METHOD parktelescope: USINT
VAR_INPUT
END_VAR
VAR
	ParkEvent:	FB_Eventlog;
	command_timeout:	TON;
END_VAR
VAR_STAT
	Stage:		USINT := 0;
	LastStage:	USINT := 101;
END_VAR
parktelescope := Stage;
command_timeout(IN := Stage < 100, PT := T#600S);
IF command_timeout.Q THEN
	error := TRUE;
	errorid := 16#20;
	Stage := 0;
END_IF
IF reset OR error THEN
	Stage := 0;
END_IF
IF isparked THEN
	Stage := 100;
END_IF
CASE Stage OF
	0: 
		gohome := 	FALSE;
		track := 	FALSE;
		goto := 	FALSE;
		slew := 	FALSE;
		IF Error THEN // emergency park
			HydraulicsControl.close_brake();
			ElevationControl.enable := FALSE;
			AzimuthElevationControl.Enable := FALSE;
			CoverControl.close := TRUE;	
			Stage := 80;
		END_IF
		Stage := 20;
	20:
		ElevationControl.position := elevation_park;
		ElevationControl.velocity := 10.0;
		ElevationControl.MoveAxis := TRUE;
		AzimuthElevationControl.position := azimuth_park;
		AzimuthElevationControl.velocity := 10;
		AzimuthElevationControl.MoveAxis := TRUE;
		IF ElevationControl.ElevationAxis.Busy AND
			AzimuthElevationControl.AzimuthAxis.Busy THEN
				Stage := 40;
		END_IF
	40:
		IF ElevationControl.ElevationAxis.MoveDone THEN
			ElevationControl.MoveAxis := FALSE;
		END_IF
		IF AzimuthElevationControl.AzimuthAxis.MoveDone THEN
			AzimuthElevationControl.MoveAxis := FALSE;
		END_IF
		IF NOT sliding THEN // all axis standstill
			Stage := 60;
		END_IF
	60:
		IF stopped THEN 
			ElevationControl.enable := FALSE;
			AzimuthElevationControl.Enable := FALSE;
			Stage := 80;
		END_IF
		
		ElevationControl.MoveAxis := FALSE;
		AzimuthElevationControl.MoveAxis := FALSE;
	80:
		IF HydraulicsControl.brake_closed THEN
			CoverControl.close := TRUE;			
		END_IF
		IF CoverControl.isclosed THEN
			Stage := 100;
		END_IF
	100:
			isparked := TRUE;
			park := FALSE;
			parktelescope := 100;
			Stage := 0;	
END_CASE
ParkEvent(Trigger := Stage > LastStage, FormatString := 'Parking progress: %s', OnMessage := USINT_TO_STRING(Stage));
LastStage := Stage;
END_METHOD

METHOD poweron : BOOL
VAR_INPUT
END_VAR
VAR
END_VAR
IF NOT Main.brake_clearing THEN
	powerfailure := TRUE;
	TCSpowerEvent.OnMessage := 'failure: brake clearing not set';
	power := FALSE;
ELSIF NOT Transformer.power_OK THEN
	powerfailure := TRUE;
	TCSpowerEvent.OnMessage := 'failure: main power failure';
	power := FALSE;
ELSIF NOT Transformer.phase_available THEN
	powerfailure := TRUE;
	TCSpowerEvent.OnMessage := 'failure: hydraulics power failure';
	power := FALSE;
ELSIF error THEN
	powerfailure := TRUE;
	TCSpowerEvent.OnMessage := 'Generic error during power on occured.';
	power := FALSE;
ELSE
	powerfailure := FALSE;		
END_IF
// COVER MUST BE OPENED FOR A SUCCESSFUL WAKE & SHAKE COMMAND!
Covercontrol.open := TRUE;

// enable elevation, enable azimuth
IF MAIN.ready AND CoverControl.isopen THEN
	ElevationControl.enable := TRUE;
	AzimuthElevationControl.enable := TRUE;
END_IF

IF ElevationControl.Ready AND NOT ElevationControl.Calibrated THEN
	ElevationControl.HomeAxis := TRUE;
END_IF

IF AzimuthElevationControl.ready AND NOT AzimuthElevationControl.calibrated THEN
	AzimuthElevationControl.HomeAxis := TRUE;
END_IF

// start calibration of focus after elevation has been calibrated
// this avoids imbalance by the M2 mirror on the elvation during its calibration

IF CoverControl.isopen AND 
	ElevationControl.Calibrated AND ElevationControl.Ready AND
	AzimuthElevationControl.calibrated AND AzimuthElevationControl.ready THEN
	power := FALSE;
	poweron := TRUE;
	isparked := FALSE;
	// slew the telescope to the home position
	gohome := TRUE;
ELSE
	poweron := FALSE;
END_IF
END_METHOD

METHOD slewtelescope : USINT
VAR_INPUT
END_VAR
VAR
	SlewEvent:	FB_Eventlog;
	command_timeout: TON;
END_VAR
VAR_STAT
	Stage:		USINT := 0;
	LastStage:	USINT := 101;
END_VAR
slewtelescope := Stage;
command_timeout(IN := Stage < 100, PT := T#600S);
IF command_timeout.Q THEN
	error := TRUE;
	errorid := 16#40;
	slew := FALSE;
	Stage := 0;
END_IF
IF reset OR error THEN
	Stage := 0;
END_IF
CASE Stage OF
	0:	
		IF ready AND stopped AND NOT busy AND NOT tracking THEN
			Stage := 25;
		END_IF
	25:
		ElevationControl.position := elevation;
		ElevationControl.velocity := 5.0;
		ElevationControl.MoveAxis := TRUE;
		AzimuthElevationControl.position := azimuth;
		AzimuthElevationControl.velocity := 10.0;
		AzimuthElevationControl.MoveAxis := TRUE;
		IF ElevationControl.ElevationAxis.Busy AND
			AzimuthElevationControl.AzimuthAxis.Busy THEN
				Stage := 50;
		END_IF
	50:
		IF ElevationControl.ElevationAxis.MoveDone THEN
			ElevationControl.MoveAxis := FALSE;
		END_IF
		
		IF AzimuthElevationControl.AzimuthAxis.MoveDone THEN
			AzimuthElevationControl.MoveAxis := FALSE;
		END_IF

		IF NOT sliding AND stopped THEN // all axis standstill
			Stage := 100;
		END_IF
	100:
		ElevationControl.MoveAxis := FALSE;
		AzimuthElevationControl.MoveAxis := FALSE;
		rightascension := rightascension_calc;
		declination := declination_calc;
		slew := FALSE;
		Stage := 0;
END_CASE
SlewEvent(Trigger := Stage > LastStage, FormatString := 'Slew progress: %s', OnMessage := USINT_TO_STRING(Stage));
LastStage := Stage;
END_METHOD

METHOD stoptelescope : BOOL
VAR_INPUT
END_VAR
ElevationControl.StopAxis := TRUE;
AzimuthElevationControl.StopAxis := TRUE;
IF stopped THEN
	ElevationControl.StopAxis := FALSE;
	AzimuthElevationControl.StopAxis := FALSE;
	stop := FALSE;
END_IF
END_METHOD

METHOD tracktelescope : BOOL
VAR_INPUT
END_VAR
// Elevation
ElevationVelocity := F_Elevationvelocity(azimuth_calc, latitude);
AzimuthVelocity := F_Azimuthvelocity(elevation_calc, azimuth_calc, latitude);
IF elevation_current < 5.0 OR elevation_current > 89.5 THEN 
	track := FALSE;
END_IF
IF azimuth_current > 440.0 THEN
	track := FALSE;
END_IF

ElevationControl.position := elevation_calc;
IF NOT ElevationControl.Tracking THEN
	ElevationControl.velocity := 10.0;
	ElevationControl.MoveAxis := TRUE;
	IF NOT ElevationControl.ElevationAxis.Busy AND ElevationControl.ElevationAxis.MoveDone THEN
		ElevationControl.MoveAxis := FALSE;
		IF ElevationControl.ElevationAxis.isTracking THEN
			ElevationControl.velocity := ElevationVelocity;
		ELSE
			ElevationControl.velocity := 3.0*ElevationVelocity;
		END_IF
		ElevationControl.velocity := ElevationVelocity;
		ElevationControl.Tracking := TRUE;
	END_IF
ELSE
	ElevationControl.velocity := ElevationVelocity;
END_IF

// Azimuth
AzimuthElevationControl.position := azimuth_calc;
IF NOT AzimuthElevationControl.Tracking THEN
	AzimuthElevationControl.velocity := 10.0;
	AzimuthElevationControl.MoveAxis := TRUE;
	IF NOT AzimuthElevationControl.AzimuthAxis.Busy AND AzimuthElevationControl.AzimuthAxis.MoveDone THEN
		AzimuthElevationControl.MoveAxis := FALSE;
		IF AzimuthElevationControl.AzimuthAxis.isTracking THEN
			AzimuthElevationControl.velocity := AzimuthVelocity;
		ELSE
			AzimuthElevationControl.velocity := 3.0*AzimuthVelocity;
		END_IF
		AzimuthElevationControl.velocity := AzimuthVelocity;
		AzimuthElevationControl.Tracking := TRUE;
	END_IF
ELSE
	AzimuthElevationControl.velocity := AzimuthVelocity;
END_IF
END_METHOD

END_PROGRAM

// ---- POUs/Function Blocks/FB_EQ2HOR2.TcPOU
FUNCTION_BLOCK FB_EQ2HOR2
VAR_INPUT
	// right ascension in degrees
	alpha: LREAL;
	// declination in degrees
	delta: LREAL;
	// longitude in degrees
	lon: LREAL;
	// latitude in degrees
	lat: LREAL;
	// Julian Days
	JD: LREAL;
END_VAR
VAR_OUTPUT
	// altitude in degrees
	alt: LREAL;
	// azimuth in degrees
	az: LREAL;
	// hour angle in degreesss
	ha: LREAL;
END_VAR
VAR
	lst: LREAL;
	// helper variables
	sinalt,
	// in radians
	phi_r, tau_r, alpha_r, delta_r: LREAL;
	// current epoch
	J_now: 		LREAL;
	// enable precession
	precess: 	BOOL := TRUE;
	// enable nutation
	nutate:		BOOL := TRUE;
	// enable abberation
	abberation:	BOOL := TRUE;
	// enable refraction correction
	refract:	BOOL := TRUE;
	// precession function block
	fbprecess: 	FB_PRECESS3;
	// nutation function block
	co_nutate: CO_NUTATE;
	// abberration function block
	fbaberration: CO_ABERRATION;
	//precessed coordinates
	alpha1, delta1, 
	d_alpha2, d_delta2, 
	d_alpha3, d_delta3:	LREAL;
END_VAR
VAR CONSTANT
	d2r:	LREAL := PI/180.0;
	r2d:	LREAL := 180.0/PI;
END_VAR

(* 
source: http://star-www.st-and.ac.uk/~fv/webnotes/chapter7.htm
https://squarewidget.com/astronomical-calculations-sidereal-time/

*)
lst := ct2lst(lon, jd) * 15.0; // lst in degrees

J_now := (JD - 2451545.0)/365.25 + 2000.0; // compute current equinox
IF precess THEN
	fbprecess( ra := alpha, dec := delta, 
	//EQUINOX1 := 2000.0, EQUINOX2 := J_now, 
	ra_precessed =>alpha1, dec_precessed => delta1);
ELSE
	alpha1 := alpha;
	delta1 := delta;	
END_IF

IF nutate THEN
	co_nutate(	jd := jd, 
				ra := alpha, 
				dec := delta, 
				d_ra => d_alpha2, 
				d_dec => d_delta2);
	alpha1 := alpha1 + d_alpha2;
	delta1 := delta1 + d_delta2;
ELSE
	d_alpha2 := 0.0;
	d_delta2 := 0.0;
END_IF

IF abberation THEN
	fbaberration(	jd := jd, 
					ra := alpha, 
					dec := delta, 
					d_ra => d_alpha3, 
					d_dec => d_delta3);
	alpha1 := alpha1 + d_alpha3;
	delta1 := delta1 + d_delta3;
ELSE
	d_alpha3 := 0.0;
	d_delta3 := 0.0;
END_IF

ha := MODABS(lst - alpha1, 360.0);

alpha_r := alpha1 * d2r;
delta_r := delta1 * d2r;
tau_r := lst*d2r - alpha_r;
phi_r := lat*d2r;

sinalt := SIN(phi_r)*SIN(delta_r) + COS(phi_r)*COS(delta_r)*COS(tau_r);
alt := ASIN(sinalt) * r2d;
IF refract THEN
	alt := alt + Refraction(alt, pressure := 770.0, temperature := 10.0);
END_IF
az := ATAN2(SIN(tau_r), SIN(phi_r)*COS(tau_r) - COS(phi_r)*TAN(delta_r)) * r2d + 180.0;

END_FUNCTION_BLOCK

// ---- POUs/Function Blocks/CO_ABERRATION.TcPOU
FUNCTION_BLOCK CO_ABERRATION
VAR_INPUT
	jd, 				// Julian Date
	ra, dec: LREAL; 	//ra and dec in degrees
	eps : LREAL := 0.0;
END_VAR
VAR_OUTPUT
	d_ra, d_dec: LREAL;
END_VAR
VAR
	sunpos: FB_SUNPOS;
	nutate: FB_NUTATE;
	sunra, sundec, sunlon,
	d_psi, d_epsilon, eps0,
	t, e, peri, cd, sd, ce, te, cp, sp, cs, ss, ca, sa, term1, term2, term3, term4: LREAL;
END_VAR
VAR CONSTANT
	d2r : LREAL := PI/180.0;
	k: LREAL := 20.49552; //constant of aberration, in arcseconds
	
END_VAR

(*
;+
;  NAME:
;     CO_ABERRATION
; PURPOSE:
;     Calculate changes to Ra and Dec due to the effect of annual aberration 
; EXPLANATION:
;      as described in Meeus, Chap 23.
; CALLING SEQUENCE:
;      co_aberration, jd, ra, dec, d_ra, d_dec, [EPS = ]
; INPUTS
;       jd      : Julian Date [scalar or vector]
;       ra, dec : Arrays (or scalars) of the ra  and dec's in degrees
;   Note: if jd is a vector, then ra and dec must either be scalars, or 
;                vectors of the same length.
;
; OUTPUTS
;       d_ra, d_dec: the corrections to ra and dec due to aberration in 
;                    arcseconds.  (These values can be added to the true RA 
;                    and dec to get the apparent position).   Note that d_ra
;                     is *not* multiplied by cos(dec), so that 
;                     apparent_ra = ra + d_ra/3600. 
; OPTIONAL INPUT KEYWORD:
;       eps : set this to the true obliquity of the ecliptic (in radians), or
;         it will be set for you if you don't know it (in that case, set it to
;                 an empty variable).
; EXAMPLE:
;   Compute the change in RA and Dec of Theta Persei (RA = 2h46m,11.331s, Dec =
;   49d20',54.54") due to aberration on 2028 Nov 13.19 TD
;
;      IDL> jdcnv,2028,11,13,.19*24,jd      ;Get Julian date
;      IDL> co_aberration,jd,ten(2,46,11.331)*15,ten(49,20,54.54),d_ra,d_dec
;
;      ==> d_ra = 30.045" (=2.003s)    d_dec = 6.697"
; NOTES:
;  These formula are from Meeus, Chapters 23.  Accuracy is much better than 1 
;   arcsecond.
;
;   The maximum deviation due to annual aberration is 20.49" and occurs when the
;   Earth velocity is perpendicular to the direction of the star.
;
; REVISION HISTORY:
;   Written, June 2002,      Chris O'Dell, U. of Wisconsin
;   Fix error with vector input   W. Landsman   June 2009
;   June 2009 update fixed case where JD was scalar but RA,Dec were vectors, but 
;     broke the case when both JD and RA,Dec were vectors Aug 2012 W. Landsman
;   Further fix when JD is 1 element vector  W. Landsman
;-
*)

T := (jd -2451545.0)/36525.0; // julian centuries from J2000 of jd.

IF EPS = 0.0 THEN
	// must calculate obliquity of ecliptic
	nutate(jd := jd, nut_long => d_psi, nut_obliq => d_epsilon); //d_psi and d_epsilon in degrees
	eps0 := ten(23,26,21.448)*3600.0 - 46.8150*T - 0.00059*EXPT(T, 2) +  0.001813*EXPT(T, 3);
	// TRUE obliquity OF the ecliptic in radians
	eps := (eps0 + d_epsilon)/3600.0*d2r; 	
END_IF

sunpos( JD := jd, RA => sunra, Dec => sundec, longmed => sunlon);

// Earth's orbital eccentricity
e := 0.016708634 - 0.000042037*T - 0.0000001267*EXPT(T, 2);
// longitude of perihelion, in degrees 
peri := 102.93735 + 1.71946*T + 0.00046*EXPT(T, 2);

//Useful Trig Functions
cd := COS(dec*d2r);		sd := SIN(dec*d2r);
ce := COS(eps); 		te := TAN(eps);
cp := COS(peri*d2r);	sp := SIN(peri*d2r);
cs := COS(sunlon*d2r);	ss := SIN(sunlon*d2r);
ca := COS(ra*d2r);		sa := SIN(ra*d2r);

term1 := (ca*cs*ce + sa*ss)/cd;
term2 := (ca*cp*ce + sa*sp)/cd;
term3 := (cs*ce*(te*cd - sa*sd) + ca*sd*ss);
term4 := (cp*ce*(te*cd - sa*sd) + ca*sd*sp);

d_ra := (-k * term1 + e*k * term2)/3600.0;
d_dec := (-k * term3 + e*k * term4)/3600.0;

END_FUNCTION_BLOCK

// ---- POUs/Functions/Refraction.TcPOU
FUNCTION Refraction : LREAL
VAR_INPUT
	// elevation in degrees
	elevation: LREAL;
	// pressure in mBar
	pressure: LREAL := 770.0;
	// temperature in Celsius
	temperature : LREAL := 10.0;
END_VAR
VAR
END_VAR
VAR CONSTANT
	d2r:	LREAL := PI/180.0;
END_VAR

// sanity checks
elevation := LIMIT(0.0, elevation, 90.0);
pressure := LIMIT(600.0, pressure, 1200.0);
temperature := LIMIT(-30.0, temperature, 40.0);
// refraction in arcmin
Refraction := 1.02 / TAN((elevation + 10.3/(elevation + 5.11)) * d2r);
Refraction := Refraction * pressure * 283.0 / (1010.0 * (273.0 + temperature));
//refraction in degrees
Refraction := Refraction / 60.0;

END_FUNCTION

// ---- POUs/Function Blocks/FB_HOR2EQ.TcPOU
FUNCTION_BLOCK FB_HOR2EQ
VAR_INPUT
	//altitude (in degrees) [scalar OR vector]
	alt: LREAL;  
	//azimuth angle (in degrees, measured EAST from NORTH, but see keyword WS below.) [scalar or vector]
	az: LREAL;
	// Julian Date [scalar or vector], double precision
	JD: 		LREAL;
	lat:		LREAL;
	lon:		LREAL;
	WS:			BOOL;
	precess:	BOOL := FALSE;
	NUTATE:		BOOL := FALSE;
	aberration:	BOOL := FALSE;
	refract:	BOOL := FALSE;
	altitude:	LREAL := 0.0;
END_VAR
VAR_OUTPUT
	// Right Ascension of object  (J2000) in degrees (FK5)
	ra: 	LREAL;
	// Declination of object (J2000) in degrees (FK5)
	dec:	LREAL;
	// hour angle (in degrees) (optional)
	ha:		LREAL;
END_VAR
VAR
	
	alt_,
	az_,
	lmst,
	J_now: LREAL;
	co_nutate: 		FB_CO_NUTATE;
	co_aberration: 	CO_ABERRATION;
	co_refract:		CO_REFRACT;
	fbprecess:		FB_PRECESS;
	altaz2hadec:	FB_ALTAZ2HADEC;
	last: LREAL;
	dra1: LREAL;
	ddec1: LREAL;
	eps: LREAL;
	d_psi: LREAL;
	dra2: LREAL;
	ddec2: LREAL;
END_VAR
VAR CONSTANT
	//d2r:	LREAL := PI/180.0;
	//r2d:	LREAL := 180.0/PI;
	//h2r:	LREAL := PI/12.0;
	h2d:	LREAL := 15.0;
END_VAR

alt_ := alt;   //do this so we don't change ra, dec arrays.
az_ := az;


//*******************************************************************************************
// Make Correction for ATMOSPHERIC REFRACTION
// (use this for visible and radio wavelengths; author is unsure about other wavelengths)
IF refract THEN 
	co_refract(	old_alt := alt, 
				altitude := altitude, 
				to_observed := TRUE, 
				new_alt => alt);
END_IF

IF WS THEN 
	az_ := az_ - 180.0;
END_IF

co_nutate(	jd := jd, 
			ra := 45.0, 
			dec := 45.0, 
			d_ra => dra1, 
			d_dec => ddec1, 
			eps => eps, 
			d_psi => d_psi);
//******************************************************************************
//Calculate LOCAL APPARENT SIDEREAL TIME
// first get local mean sidereal time (lmst)
// get LST (in hours) - note:this is indep of tzone since giving jd
lmst := ct2lst( lon, jd);
// convert LMST TO degrees (btw, THIS is the RA OF the zenith)
lmst := lmst*h2d;
// calculate local APPARENT sidereal time (last)
// ADD correction in degrees
last := lmst + d_psi *COS(eps)/3600.0 ; 

//****************************************************************************
// Now do the spherical trig to get APPARENT Hour Angle [degrees], and
// declination [degrees].
altaz2hadec( alt := alt_, az := az_, lat := lat, ha => ha, dec => dec);

// Find Right Ascension (in degrees, from 0 to 360.)
 ra := MODABS(last - ha + 360.0, 360.0);



//*****************************************************************************
// calculate NUTATION and ABERRATION Corrections to Ra-Dec
IF NUTATE THEN
	co_nutate(	jd := jd, 
			ra := ra, 
			dec := dec, 
			d_ra => dra1, 
			d_dec => ddec1, 
			eps => eps, 
			d_psi => d_psi);
ELSE
	dra1 := 0.0;
	ddec1 := 0.0;	
END_IF
IF aberration THEN
	co_aberration(	jd := jd, 
				ra := ra, 
				dec := dec, 
				d_ra => dra2, 
				d_dec => ddec2, 
				eps := eps);
ELSE
	dra2 := 0.0;
	ddec2 := 0.0;	
END_IF
//******************************************************************************
// Make Nutation and Aberration Corrections (if wanted)

ra := ra - (dra1 + dra2)/3600.0;
dec := dec - (ddec1 + ddec2)/3600.0;
 //compute current equinox
J_now := (JD - 2451545.0)/365.25 + 2000.0 ;

//*****************************************************************************
// PRECESS coordinates to current date
// (uses astro lib procedure PRECESS.pro)

IF precess THEN 
	fbprecess( ra := ra, dec := dec, 
	EQUINOX1 := J_now, EQUINOX2 := 2000.0, // bugfix from randnotizlukas
	ra_precessed =>ra, dec_precessed => dec);                   
END_IF

END_FUNCTION_BLOCK

// ---- POUs/TelescopeAuxiliary.TcPOU
PROGRAM TelescopeAuxiliary
VAR
	MQTTTimer : TON := (PT:=T#5S);
	cycle:	USINT;
	FBReadPressure : FB_ReadAdsSymByName;
	FBReadTemperature: FB_ReadAdsSymByName;
	// EL3064-1
	raw_dewar_pressure		AT%I*: INT;
	pressure_voltage:	REAL;
	dewar_warning_trigger: SR;
	dewar_error_trigger: SR;
	DewarWarning, DewarError: FB_EventLog;
END_VAR
VAR_OUTPUT
	// BT9 mirror
	temperature_mirror2:	REAL;
	// BT10
	temperature_mirror1:	REAL;
	pressure:		REAL;
	temperature:	REAL;
	dewar_pressure:	REAL;
	dewar_pressure_atm: REAL;
END_VAR

temperature_mirror1 := F_YREAL(GVL_Telescope.temperature_mirror1, 0, 32767, 0.0, 100.0);
temperature_mirror2 := F_YREAL(GVL_Telescope.temperature_mirror1, 0, 32767, -50.0, 100.0);


cycle := cycle MOD 8;
FBReadPressure(
	bRead := cycle MOD 10 = 1,
	sNetId := '5.40.71.146.1.1',
	sVarName := 'Environment.Pressure',
	nDestAddr := ADR(pressure),
	nLen := SIZEOF(pressure),
 	eComMode := eAdsComModeFastCom
	);
FBReadTemperature(
	bRead := cycle MOD 10 = 4,
	sNetId := '5.40.71.146.1.1',
	sVarName := 'Environment.Temperature1',
	nDestAddr := ADR(temperature),
	nLen := SIZEOF(temperature),
 	eComMode := eAdsComModeFastCom
	);
IF NOT (FBReadPressure.bBusy OR FBReadPressure.bError) AND 
   NOT (FBReadTemperature.bBusy OR FBReadTemperature.bError) THEN
	cycle := cycle + 1;
END_IF

pressure_voltage := F_YREAL(raw_dewar_pressure, 0, 32767, 0.0, 10.0);
dewar_pressure := LREAL_TO_REAL(EXPT(10.0, F_YREAL(pressure_voltage, 2.0, 10.0, -9.0, 3.0)));
dewar_pressure_atm := LREAL_TO_REAL(EXPT(10.0, F_YREAL(pressure_voltage, 2.0, 10.0, -7.0, 5.0)));

dewar_warning_trigger(SET1 := dewar_pressure_atm > 1E-6, RESET := dewar_pressure_atm < 5E-7);
dewar_error_trigger(SET1 := dewar_pressure_atm > 1E-5, RESET := dewar_pressure_atm < 1E-6);

DewarWarning(Trigger := dewar_warning_trigger.Q1,
				Level := ADSLOG_MSGTYPE_WARN,
				FormatString := '%s',
				OnMessage := 'Dewar pressure is above nominal.',
				OffMessage := 'Dewar pressure is nominal.');

DewarError(Trigger := dewar_error_trigger.Q1,
				Level := ADSLOG_MSGTYPE_ERROR,
				FormatString := '%s',
				OnMessage := 'Dewar pressure is critical!');


MQTTTimer(IN:=TRUE);
IF MQTTTimer.Q THEN // publish new payload every second

	MAIN.MQTTClient.Publish('telescope', 'dome', 'Mirror1Temperature',	LREAL_TO_FMTSTR(temperature_mirror1, 2, TRUE));
	//MAIN.MQTTClient.Publish('telescope', 'dome', 'Mirror2Temperature',	LREAL_TO_FMTSTR(temperature_mirror2, 2, TRUE));
	MAIN.MQTTClient.Publish('telescope', 'dome', 'DewarPressureVoltage', LREAL_TO_FMTSTR(pressure_voltage, 3, TRUE));
	MAIN.MQTTClient.Publish('telescope', 'dome', 'DewarPressure', LREAL_TO_FMTSTR(dewar_pressure_atm, 9, TRUE));
	
	MQTTTimer(IN:=FALSE);

END_IF

END_PROGRAM

// ---- POUs/Functions/PointingModelAzimuth.TcPOU
FUNCTION PointingModelAzimuth : LREAL
// https://aro.as.arizona.edu/~aro/12_obs_manual/pdfs/Appendix_A_Rev_2.pdf
VAR_INPUT
	// current azimuth of telescope in degrees
	azimuth: LREAL;
	// current elevation of telescope in degrees
	elevation: LREAL;
	// azimuth encoder zero offset
	AOFF: 	LREAL;
	// collimation error of the electromagnetic axis
	BNP:	LREAL;
	// azimuth axis offset/misalignment north-south
	AN_A:	LREAL;
	// azimuth axis offset/misalignment east-west,
	AE_A:	LREAL;
	// Non-perpendicularity between the mount azimuth and elevation axes
	NPAE:	LREAL;
END_VAR
VAR
	tan_elevation:	LREAL;
	cos_elevation:	LREAL;
END_VAR
VAR CONSTANT
	d2r:	LREAL := PI/180.0;
	//r2d:	LREAL := 180.0/PI;
END_VAR

IF elevation<89.9 THEN
	tan_elevation := TAN(elevation * d2r);
	cos_elevation := COS(elevation * d2r);
ELSE // clamp values so that we do not run into DIV by zero or overflow
	tan_elevation := 572.9572133543033;
	cos_elevation := 0.0017453283658982613;
END_IF

//d(az)=AOFF-BNP/cos(el)+NPAE*tan(el)+AAN*sin(az)*tan(el)-AAE*cos(az)*tan(el)

PointingModelAzimuth := AOFF - BNP/cos_elevation + AN_A*SIN(azimuth * d2r)*tan_elevation - AE_A*COS(azimuth * d2r)*tan_elevation + NPAE*tan_elevation;

END_FUNCTION

// ---- POUs/Function Blocks/FB_EL3443.TcPOU
(*  This function block calls up the variant values supplied by the EL3443 terminal. The multiplexer channels of the terminal are queried by the use of selectors.
    Due to the multiplexing of the values in the variant values, reading the terminal information requires several PLC cycles.
    In contrast, values that can be retrieved via the process image are output cyclically. 
    
    To use the function block:
    ▪ the predefined PDO assignment "Default + Variant" must be selected for the terminal under "Process data".
    
    ▪ Then the PLC data type (structure from the process data, MDP5001_341_7FF5D4A6) must be activated in the "PLC" tab of the terminal.
    
    ▪ After creating the data type, the PLC project must be rebuilt.
    
    ▪ Finally, the terminal must be linked to the function block on the "PLC" tab*)

{attribute 'no-analysis'}  
{attribute 'hide_all_locals'}   
FUNCTION_BLOCK FB_EL3443
VAR_INPUT
    bEnable : BOOL; //Enables the Variant values to be queried using the multiplexer functions of the block
	
    stEL3443_IO : MDP5001_341_7FF5D4A6; //External data type that can be generated within the terminal on the PLC tab
END_VAR

VAR_OUTPUT
    stStatusTotal 	 : ST_EL3443_StatusTotal; //General cyclical process data
    stStatusPhase_L1 : ST_EL3443_StatusLx; //Phase L1 specific cyclical process data 
    stStatusPhase_L2 : ST_EL3443_StatusLx; //Phase L2 specific cyclical process data
    stStatusPhase_L3 : ST_EL3443_StatusLx; //Phase L3 specific cyclical process data
    stVariantValues	 : ST_EL3443_VariantValues; //Variant Values (non-cyclical values). Due to the multiplexing of the values in the Variant Values, the reading of the terminal information requires several PLC cycles.
    
    bError : BOOL; //Becomes TRUE as soon as an error situation occurs.
END_VAR

VAR    
    {attribute 'no_copy'}
	astEL3443MuxReal_Ch1: ARRAY [0..nARRAYSIZEMUXREAL] OF ST_EL3443_MUX_REAL; //Structure for the (Real) Multiplexer Channel 1 contains the selector and a reference to the corresponding memory location
    {attribute 'no_copy'}
    astEL3443MuxReal_Ch2: ARRAY [0..nARRAYSIZEMUXREAL] OF ST_EL3443_MUX_REAL; //Structure for the (Real) Multiplexer Channel 2 contains the selector and a reference to the corresponding memory location
    {attribute 'no_copy'}
    astEL3443MuxReal_Ch3: ARRAY [0..nARRAYSIZEMUXREAL] OF ST_EL3443_MUX_REAL; //Structure for the (Real) Multiplexer Channel 3 contains the selector and a reference to the corresponding memory location   
    {attribute 'no_copy'}
	stEL3443MuxUlint_Ch4: ARRAY [0..nARRAYSIZEMUXULINT] OF ST_EL3443_MUX_ULINT; //Structure for the (ULINT/LINT) multiplexer channel 4 contains the selector and a pointer to the corresponding memory location
    
    {attribute 'no_copy'}
    bInit : BOOL; //Flag to indicate the initialised state of the function block
    nMuxRealState : INT := 0; //Position der Multplexer-Abfragen (Channel 1-3 (REAL))
    nCounterNotRepliedMuxReal : INT; //Number of cycles in which the multiplexer has not responded
    nMuxUlintState : INT := 0; //Position der Multplexer-Abfragen (Channel 4 (ULINT))
    nCounterNotRepliedMuxUlint : INT; //Number of cycles in which the multiplexer has not responded
    
        
    {attribute 'no_copy'}
    nNumberOfSelectorsCh1 : UINT; //number of selectors in channel 1  
    {attribute 'no_copy'}
    nNumberOfSelectorsCh2 : UINT; //number of selectors in channel 2   
    {attribute 'no_copy'}
    nNumberOfSelectorsCh3 : UINT; //number of selectors in channel 3 
    {attribute 'no_copy'}
    nNumberOfSelectorsCh4 : UINT; //number of selectors in channel 4    
END_VAR

VAR CONSTANT 
    nARRAYSIZEMUXREAL  : INT := 122; //Array size of the REAL multiplexer channel
    nARRAYSIZEMUXULINT : INT := 74; //Array size of the ULINT multiplexer channel
    nERROR_NOT_REPLIED : INT := 10; //Maximum number of cycles the multiplexer may use before the error output is set 
END_VAR

//The output bError is set if the block is enabled and one of the multiplexer channels does not respond
bError := bEnable AND ((nCounterNotRepliedMuxUlint >= nERROR_NOT_REPLIED) OR (nCounterNotRepliedMuxReal >= nERROR_NOT_REPLIED));

IF bEnable THEN
      
    IF NOT bInit THEN
        bInit := TRUE;
        Initialize();
    END_IF
    
    //===================================================================================================================================
    // Multiplexer channels 1-3 (REAL)
    
    //comparison of the transmitting and receiving selectors 
    IF astEL3443MuxReal_Ch1[nMuxRealState].nSelector = stEL3443_IO.MDP5001_341_Input.MDP5001_341_Total_Variant_Value_In_Index_1_REAL AND
       astEL3443MuxReal_Ch2[nMuxRealState].nSelector = stEL3443_IO.MDP5001_341_Input.MDP5001_341_Total_Variant_Value_In_Index_2_REAL AND 
       astEL3443MuxReal_Ch3[nMuxRealState].nSelector = stEL3443_IO.MDP5001_341_Input.MDP5001_341_Total_Variant_Value_In_Index_3_REAL THEN
        
    
        //assignment of the received values to the referenced references
        IF __ISVALIDREF(astEL3443MuxReal_Ch1[nMuxRealState].fValueRef) THEN
            astEL3443MuxReal_Ch1[nMuxRealState].fValueRef := stEL3443_IO.MDP5001_341_Input.MDP5001_341_Total_Variant_Value_In_Value_1_REAL;
        END_IF
        IF __ISVALIDREF(astEL3443MuxReal_Ch2[nMuxRealState].fValueRef) THEN
            astEL3443MuxReal_Ch2[nMuxRealState].fValueRef := stEL3443_IO.MDP5001_341_Input.MDP5001_341_Total_Variant_Value_In_Value_2_REAL;
        END_IF
        IF __ISVALIDREF(astEL3443MuxReal_Ch3[nMuxRealState].fValueRef) THEN
            astEL3443MuxReal_Ch3[nMuxRealState].fValueRef := stEL3443_IO.MDP5001_341_Input.MDP5001_341_Total_Variant_Value_In_Value_3_REAL;
        END_IF
       
       //selection of the new selector group
       nMuxRealState := nMuxRealState + 1;
     
       IF nMuxRealState > nARRAYSIZEMUXREAL THEN
         nMuxRealState := 0;  
       END_IF
       
       nCounterNotRepliedMuxReal := 0;
    ELSIF
        stEL3443_IO.MDP5001_341_Input.MDP5001_341_Total_Variant_Value_In_Index_1_REAL = E_EL3443_Phase.Error_INDEX_Not_Valid OR    
        stEL3443_IO.MDP5001_341_Input.MDP5001_341_Total_Variant_Value_In_Index_2_REAL = E_EL3443_Phase.Error_INDEX_Not_Valid OR 
        stEL3443_IO.MDP5001_341_Input.MDP5001_341_Total_Variant_Value_In_Index_3_REAL = E_EL3443_Phase.Error_INDEX_Not_Valid THEN
    
        nCounterNotRepliedMuxReal := MIN(nCounterNotRepliedMuxReal + 1,nERROR_NOT_REPLIED);
    ELSE
        nCounterNotRepliedMuxReal := MIN(nCounterNotRepliedMuxReal + 1,nERROR_NOT_REPLIED); 
    END_IF
       
    // transfer of the selectors to the process image 
    stEL3443_IO.MDP5001_341_Output.MDP5001_341_Total_Variant_Value_Out_Index_1_REAL := astEL3443MuxReal_Ch1[nMuxRealState].nSelector;
    stEL3443_IO.MDP5001_341_Output.MDP5001_341_Total_Variant_Value_Out_Index_2_REAL := astEL3443MuxReal_Ch2[nMuxRealState].nSelector;
    stEL3443_IO.MDP5001_341_Output.MDP5001_341_Total_Variant_Value_Out_Index_3_REAL := astEL3443MuxReal_Ch3[nMuxRealState].nSelector;
    
    //===================================================================================================================================
    // Multiplexer channels 4 (ULINT)
    
    //comparison of the transmitting and receiving selector
    IF stEL3443MuxUlint_Ch4[nMuxUlintState].nSelector = stEL3443_IO.MDP5001_341_Input.MDP5001_341_Total_Variant_Value_In_Index_4_ULINT THEN
        
        //assigns the received values to the assigned pointer address.
        IF stEL3443MuxUlint_Ch4[nMuxUlintState].nValueRef <> 0 THEN
            stEL3443MuxUlint_Ch4[nMuxUlintState].nValueRef^ := stEL3443_IO.MDP5001_341_Input.MDP5001_341_Total_Variant_Value_In_Value_4_ULINT;
        END_IF
        
    //selection of the new selector group
       nMuxUlintState := nMuxUlintState + 1;
     
       IF nMuxUlintState > nARRAYSIZEMUXULINT THEN
         nMuxUlintState := 0;  
       END_IF
       
       nCounterNotRepliedMuxUlint := 0;
    ELSIF stEL3443_IO.MDP5001_341_Input.MDP5001_341_Total_Variant_Value_In_Index_4_ULINT = E_EL3443_Phase.Error_INDEX_Not_Valid THEN
    
        nCounterNotRepliedMuxUlint := MIN(nCounterNotRepliedMuxUlint + 1, nERROR_NOT_REPLIED);
    ELSE
        nCounterNotRepliedMuxUlint := MIN(nCounterNotRepliedMuxUlint + 1, nERROR_NOT_REPLIED);  
    END_IF
    
    // transfer of the selectors to the process image
    stEL3443_IO.MDP5001_341_Output.MDP5001_341_Total_Variant_Value_Out_Index_4_ULINT := stEL3443MuxUlint_Ch4[nMuxUlintState].nSelector;
END_IF

//===================================================================================================================================
// Update the cyclic outputs
// Transfer of process data to PLC common data types. Status total.
stStatusTotal.bStatus_System_State :=                       stEL3443_IO.MDP5001_341_Input.MDP5001_341_Total_Status_System_State;
stStatusTotal.bStatus_Grid_Direction :=                     stEL3443_IO.MDP5001_341_Input.MDP5001_341_Total_Status_Grid_Direction;
stStatusTotal.bStatus_Frequency_Guard_Warning :=            stEL3443_IO.MDP5001_341_Input.MDP5001_341_Total_Status_Frequency_Guard_Warning;
stStatusTotal.bStatus_Frequency_Guard_Error :=              stEL3443_IO.MDP5001_341_Input.MDP5001_341_Total_Status_Frequency_Guard_Error;
stStatusTotal.bStatus_Neutral_Current_Guard_Warning :=      stEL3443_IO.MDP5001_341_Input.MDP5001_341_Total_Status_Neutral_Current_Guard_Warning;
stStatusTotal.bStatus_Neutral_Current_Guard_Error :=        stEL3443_IO.MDP5001_341_Input.MDP5001_341_Total_Status_Neutral_Current_Guard_Error;
stStatusTotal.bStatus_Active_Power_Guard_Warning :=         stEL3443_IO.MDP5001_341_Input.MDP5001_341_Total_Status_Active_Power_Guard_Warning;    
stStatusTotal.bStatus_Active_Power_Guard_Error :=           stEL3443_IO.MDP5001_341_Input.MDP5001_341_Total_Status_Active_Power_Guard_Error;
stStatusTotal.bStatus_Apparent_Power_Guard_Warning :=       stEL3443_IO.MDP5001_341_Input.MDP5001_341_Total_Status_Apparent_Power_Guard_Warning;
stStatusTotal.bStatus_Apparent_Power_Guard_Error :=         stEL3443_IO.MDP5001_341_Input.MDP5001_341_Total_Status_Apparent_Power_Guard_Error; 
stStatusTotal.bStatus_Power_Quality_Guard_Warning :=        stEL3443_IO.MDP5001_341_Input.MDP5001_341_Total_Status_Power_Quality_Guard_Warning; 
stStatusTotal.bStatus_Power_Quality_Guard_Error :=          stEL3443_IO.MDP5001_341_Input.MDP5001_341_Total_Status_Power_Quality_Guard_Error; 
stStatusTotal.bStatus_TxPDO_State :=                        stEL3443_IO.MDP5001_341_Input.MDP5001_341_Total_Status_TxPDO_State; 
stStatusTotal.bStatus_TxPDO_Toggle :=                       stEL3443_IO.MDP5001_341_Input.MDP5001_341_Total_Status_TxPDO_Toggle; 
stStatusTotal.fStatus_Power_Quality_Factor :=               stEL3443_IO.MDP5001_341_Input.MDP5001_341_Total_Status_Power_Quality_Factor; 
stStatusTotal.fBasic_Frequency :=                           stEL3443_IO.MDP5001_341_Input.MDP5001_341_Total_Basic_Frequency; 
stStatusTotal.fBasic_Power_Factor :=                        stEL3443_IO.MDP5001_341_Input.MDP5001_341_Total_Basic_Power_Factor; 
stStatusTotal.fBasic_Calculated_Neutral_Line_Current :=		stEL3443_IO.MDP5001_341_Input.MDP5001_341_Total_Basic_Calculated_Neutral_Line_Current;

//Transfer of process data to PLC common data types. Status phase L1.
stStatusPhase_L1.bStatus_Voltage_Sign_Bit  :=               stEL3443_IO.MDP5001_341_Input.MDP5001_341_L1_Status_Voltage_Sign_Bit;
stStatusPhase_L1.bStatus_Overvoltage  :=                    stEL3443_IO.MDP5001_341_Input.MDP5001_341_L1_Status_Overvoltage;
stStatusPhase_L1.bStatus_Overcurrent  :=                    stEL3443_IO.MDP5001_341_Input.MDP5001_341_L1_Status_Overcurrent;
stStatusPhase_L1.bStatus_Inaccurate_Voltage  :=             stEL3443_IO.MDP5001_341_Input.MDP5001_341_L1_Status_Inaccurate_Voltage;
stStatusPhase_L1.bStatus_Inaccurate_Current  :=             stEL3443_IO.MDP5001_341_Input.MDP5001_341_L1_Status_Inaccurate_Current;
stStatusPhase_L1.bStatus_Voltage_Guard_Warning  :=          stEL3443_IO.MDP5001_341_Input.MDP5001_341_L1_Status_Voltage_Guard_Warning;
stStatusPhase_L1.bStatus_Voltage_Guard_Error  :=            stEL3443_IO.MDP5001_341_Input.MDP5001_341_L1_Status_Voltage_Guard_Error;
stStatusPhase_L1.bStatus_Current_Guard_Warning  :=          stEL3443_IO.MDP5001_341_Input.MDP5001_341_L1_Status_Current_Guard_Warning;
stStatusPhase_L1.bStatus_Current_Guard_Error  :=            stEL3443_IO.MDP5001_341_Input.MDP5001_341_L1_Status_Current_Guard_Error;
stStatusPhase_L1.bStatus_TxPDO_Toggle  :=                   stEL3443_IO.MDP5001_341_Input.MDP5001_341_L1_Status_TxPDO_Toggle;
stStatusPhase_L1.fBasic_Voltage  :=                         stEL3443_IO.MDP5001_341_Input.MDP5001_341_L1_Basic_Voltage;
stStatusPhase_L1.fBasic_Current  :=                         stEL3443_IO.MDP5001_341_Input.MDP5001_341_L1_Basic_Current;
stStatusPhase_L1.fPower_Active_Power  :=                    stEL3443_IO.MDP5001_341_Input.MDP5001_341_L1_Power_Active_Power;
stStatusPhase_L1.fPower_Apparent_Power  :=                  stEL3443_IO.MDP5001_341_Input.MDP5001_341_L1_Power_Apparent_Power;
stStatusPhase_L1.fPower_Reactive_Power  :=                  stEL3443_IO.MDP5001_341_Input.MDP5001_341_L1_Power_Reactive_Power;
stStatusPhase_L1.fPower_Power_Factor  :=                    stEL3443_IO.MDP5001_341_Input.MDP5001_341_L1_Power_Power_Factor;
stStatusPhase_L1.nTiming_Voltage_Last_Zero_Crossing :=      stEL3443_IO.MDP5001_341_Input.MDP5001_341_L1_Timing_Voltage_Last_Zero_Crossing;

//Transfer of process data to PLC common data types. Status phase L2.
stStatusPhase_L2.bStatus_Voltage_Sign_Bit  :=               stEL3443_IO.MDP5001_341_Input.MDP5001_341_L2_Status_Voltage_Sign_Bit;
stStatusPhase_L2.bStatus_Overvoltage  :=                    stEL3443_IO.MDP5001_341_Input.MDP5001_341_L2_Status_Overvoltage;
stStatusPhase_L2.bStatus_Overcurrent  :=                    stEL3443_IO.MDP5001_341_Input.MDP5001_341_L2_Status_Overcurrent;        
stStatusPhase_L2.bStatus_Inaccurate_Voltage  :=             stEL3443_IO.MDP5001_341_Input.MDP5001_341_L2_Status_Inaccurate_Voltage;		
stStatusPhase_L2.bStatus_Inaccurate_Current  :=             stEL3443_IO.MDP5001_341_Input.MDP5001_341_L2_Status_Inaccurate_Current;		
stStatusPhase_L2.bStatus_Voltage_Guard_Warning  :=          stEL3443_IO.MDP5001_341_Input.MDP5001_341_L2_Status_Voltage_Guard_Warning;		
stStatusPhase_L2.bStatus_Voltage_Guard_Error  :=            stEL3443_IO.MDP5001_341_Input.MDP5001_341_L2_Status_Voltage_Guard_Error;		
stStatusPhase_L2.bStatus_Current_Guard_Warning  :=          stEL3443_IO.MDP5001_341_Input.MDP5001_341_L2_Status_Current_Guard_Warning;		
stStatusPhase_L2.bStatus_Current_Guard_Error  :=            stEL3443_IO.MDP5001_341_Input.MDP5001_341_L2_Status_Current_Guard_Error;		
stStatusPhase_L2.bStatus_TxPDO_Toggle  :=                   stEL3443_IO.MDP5001_341_Input.MDP5001_341_L2_Status_TxPDO_Toggle;		
stStatusPhase_L2.fBasic_Voltage  :=                         stEL3443_IO.MDP5001_341_Input.MDP5001_341_L2_Basic_Voltage;		
stStatusPhase_L2.fBasic_Current  :=                         stEL3443_IO.MDP5001_341_Input.MDP5001_341_L2_Basic_Current;		
stStatusPhase_L2.fPower_Active_Power  :=                    stEL3443_IO.MDP5001_341_Input.MDP5001_341_L2_Power_Active_Power;		
stStatusPhase_L2.fPower_Apparent_Power  :=                  stEL3443_IO.MDP5001_341_Input.MDP5001_341_L2_Power_Apparent_Power;		
stStatusPhase_L2.fPower_Reactive_Power  :=                  stEL3443_IO.MDP5001_341_Input.MDP5001_341_L2_Power_Reactive_Power;		
stStatusPhase_L2.fPower_Power_Factor  :=                    stEL3443_IO.MDP5001_341_Input.MDP5001_341_L2_Power_Power_Factor;
stStatusPhase_L2.nTiming_Voltage_Last_Zero_Crossing :=      stEL3443_IO.MDP5001_341_Input.MDP5001_341_L2_Timing_Voltage_Last_Zero_Crossing;
		
//Transfer of process data to PLC common data types. Status phase L3.		
stStatusPhase_L3.bStatus_Voltage_Sign_Bit  :=               stEL3443_IO.MDP5001_341_Input.MDP5001_341_L3_Status_Voltage_Sign_Bit;		
stStatusPhase_L3.bStatus_Overvoltage  :=                    stEL3443_IO.MDP5001_341_Input.MDP5001_341_L3_Status_Overvoltage;                                             
stStatusPhase_L3.bStatus_Overcurrent  :=                    stEL3443_IO.MDP5001_341_Input.MDP5001_341_L3_Status_Overcurrent;
stStatusPhase_L3.bStatus_Inaccurate_Voltage  :=             stEL3443_IO.MDP5001_341_Input.MDP5001_341_L3_Status_Inaccurate_Voltage;
stStatusPhase_L3.bStatus_Inaccurate_Current  :=             stEL3443_IO.MDP5001_341_Input.MDP5001_341_L3_Status_Inaccurate_Current;
stStatusPhase_L3.bStatus_Voltage_Guard_Warning  :=          stEL3443_IO.MDP5001_341_Input.MDP5001_341_L3_Status_Voltage_Guard_Warning;
stStatusPhase_L3.bStatus_Voltage_Guard_Error  :=            stEL3443_IO.MDP5001_341_Input.MDP5001_341_L3_Status_Voltage_Guard_Error;
stStatusPhase_L3.bStatus_Current_Guard_Warning  :=          stEL3443_IO.MDP5001_341_Input.MDP5001_341_L3_Status_Current_Guard_Warning;
stStatusPhase_L3.bStatus_Current_Guard_Error  :=            stEL3443_IO.MDP5001_341_Input.MDP5001_341_L3_Status_Current_Guard_Error;
stStatusPhase_L3.bStatus_TxPDO_Toggle  :=                   stEL3443_IO.MDP5001_341_Input.MDP5001_341_L3_Status_TxPDO_Toggle;
stStatusPhase_L3.fBasic_Voltage  :=                         stEL3443_IO.MDP5001_341_Input.MDP5001_341_L3_Basic_Voltage;
stStatusPhase_L3.fBasic_Current  :=                         stEL3443_IO.MDP5001_341_Input.MDP5001_341_L3_Basic_Current;
stStatusPhase_L3.fPower_Active_Power  :=                    stEL3443_IO.MDP5001_341_Input.MDP5001_341_L3_Power_Active_Power;
stStatusPhase_L3.fPower_Apparent_Power  :=                  stEL3443_IO.MDP5001_341_Input.MDP5001_341_L3_Power_Apparent_Power;
stStatusPhase_L3.fPower_Reactive_Power  :=                  stEL3443_IO.MDP5001_341_Input.MDP5001_341_L3_Power_Reactive_Power;
stStatusPhase_L3.fPower_Power_Factor  :=                    stEL3443_IO.MDP5001_341_Input.MDP5001_341_L3_Power_Power_Factor;
stStatusPhase_L3.nTiming_Voltage_Last_Zero_Crossing :=      stEL3443_IO.MDP5001_341_Input.MDP5001_341_L3_Timing_Voltage_Last_Zero_Crossing;

(* This method initializes the lookup table and establishes a connection between selector index and variable by references. *)
METHOD PRIVATE Initialize : HRESULT
VAR
    nPhase : INT; // Three-phase
    stEL3443MuxReal : REFERENCE TO ARRAY [0..nARRAYSIZEMUXREAL] OF ST_EL3443_MUX_REAL;
    nNumberOfSelector : REFERENCE TO UINT;
    nOFFSET : UINT;
    i : UINT;
END_VAR
// - The process data of phases L1, L2 and L3 are distributed to the three REAL multiplexers. (Channel1 = L1, Channel2 = L2 ...)
// - The ULINT multiplexer is initialized with data from all three phases.
FOR nPhase := 1 TO 3 DO
    
    // Selection of the structures, selector counters and offset based on the phase
    CASE nPhase OF
    1: // Phase L1
       stEL3443MuxReal REF= astEL3443MuxReal_Ch1;
       nNumberOfSelector REF= nNumberOfSelectorsCh1;
       nOFFSET := E_EL3443_Phase.nPhaseL1_OFFSET;  
    2: // Phase L2 
       stEL3443MuxReal REF= astEL3443MuxReal_Ch2;
       nNumberOfSelector REF= nNumberOfSelectorsCh2;
       nOFFSET := E_EL3443_Phase.nPhaseL2_OFFSET; 
    3: // Phase L3 
       stEL3443MuxReal REF= astEL3443MuxReal_Ch3;
       nNumberOfSelector REF= nNumberOfSelectorsCh3;
       nOFFSET := E_EL3443_Phase.nPhaseL3_OFFSET;
    ELSE
       EXIT;   
	END_CASE
    
    // Initializing the REAL multiplexers on channels 1 to 3
    InitSelectorReal(stEL3443MuxReal, nNumberOfSelector, stVariantValues.astLx[nPhase].fU_RMS,         nOFFSET, E_EL3443_Phase.U_RMS         );
    InitSelectorReal(stEL3443MuxReal, nNumberOfSelector, stVariantValues.astLx[nPhase].fU_peak,        nOFFSET, E_EL3443_Phase.U_peak        );
    InitSelectorReal(stEL3443MuxReal, nNumberOfSelector, stVariantValues.astLx[nPhase].fU_RMS_Minimum, nOFFSET, E_EL3443_Phase.U_RMS_Minimum);
    InitSelectorReal(stEL3443MuxReal, nNumberOfSelector, stVariantValues.astLx[nPhase].fU_RMS_Maximum, nOFFSET, E_EL3443_Phase.U_RMS_Maximum);
    InitSelectorReal(stEL3443MuxReal, nNumberOfSelector, stVariantValues.astLx[nPhase].fULL,           nOFFSET, E_EL3443_Phase.ULL          );
    InitSelectorReal(stEL3443MuxReal, nNumberOfSelector, stVariantValues.astLx[nPhase].fI_RMS,         nOFFSET, E_EL3443_Phase.I_RMS        );
    InitSelectorReal(stEL3443MuxReal, nNumberOfSelector, stVariantValues.astLx[nPhase].fI_peak,        nOFFSET, E_EL3443_Phase.I_peak       ); 
    InitSelectorReal(stEL3443MuxReal, nNumberOfSelector, stVariantValues.astLx[nPhase].fI_RMS_Minimum, nOFFSET, E_EL3443_Phase.I_RMS_Minimum );
    InitSelectorReal(stEL3443MuxReal, nNumberOfSelector, stVariantValues.astLx[nPhase].fI_RMS_Maximum, nOFFSET, E_EL3443_Phase.I_RMS_Maximum );
    InitSelectorReal(stEL3443MuxReal, nNumberOfSelector, stVariantValues.astLx[nPhase].fFrequency,     nOFFSET, E_EL3443_Phase.Frequency     );
    InitSelectorReal(stEL3443MuxReal, nNumberOfSelector, stVariantValues.astLx[nPhase].fPhi,           nOFFSET, E_EL3443_Phase.Phi,          );
    InitSelectorReal(stEL3443MuxReal, nNumberOfSelector, stVariantValues.astLx[nPhase].fCOS_phi,       nOFFSET, E_EL3443_Phase.Cos_phi       );
    InitSelectorReal(stEL3443MuxReal, nNumberOfSelector, stVariantValues.astLx[nPhase].fPower_Factor,  nOFFSET, E_EL3443_Phase.Power_Factor  );
    InitSelectorReal(stEL3443MuxReal, nNumberOfSelector, stVariantValues.astLx[nPhase].fP,             nOFFSET, E_EL3443_Phase.P             );
    InitSelectorReal(stEL3443MuxReal, nNumberOfSelector, stVariantValues.astLx[nPhase].fPavg,          nOFFSET, E_EL3443_Phase.Pavg          );
    InitSelectorReal(stEL3443MuxReal, nNumberOfSelector, stVariantValues.astLx[nPhase].fPmin,          nOFFSET, E_EL3443_Phase.Pmin          );
    InitSelectorReal(stEL3443MuxReal, nNumberOfSelector, stVariantValues.astLx[nPhase].fPmax,          nOFFSET, E_EL3443_Phase.Pmax          );
    InitSelectorReal(stEL3443MuxReal, nNumberOfSelector, stVariantValues.astLx[nPhase].fS,             nOFFSET, E_EL3443_Phase.S_            );
    InitSelectorReal(stEL3443MuxReal, nNumberOfSelector, stVariantValues.astLx[nPhase].fSavg,          nOFFSET, E_EL3443_Phase.Savg          );
    InitSelectorReal(stEL3443MuxReal, nNumberOfSelector, stVariantValues.astLx[nPhase].fSmin,          nOFFSET, E_EL3443_Phase.Smin          );
    InitSelectorReal(stEL3443MuxReal, nNumberOfSelector, stVariantValues.astLx[nPhase].fSmax,          nOFFSET, E_EL3443_Phase.Smax          );
    InitSelectorReal(stEL3443MuxReal, nNumberOfSelector, stVariantValues.astLx[nPhase].fQ,             nOFFSET, E_EL3443_Phase.Q             );
    InitSelectorReal(stEL3443MuxReal, nNumberOfSelector, stVariantValues.astLx[nPhase].fQavg,          nOFFSET, E_EL3443_Phase.Qavg          );
    InitSelectorReal(stEL3443MuxReal, nNumberOfSelector, stVariantValues.astLx[nPhase].fQmin,          nOFFSET, E_EL3443_Phase.Qmin          );
    InitSelectorReal(stEL3443MuxReal, nNumberOfSelector, stVariantValues.astLx[nPhase].fQmax,          nOFFSET, E_EL3443_Phase.Qmax          );
    InitSelectorReal(stEL3443MuxReal, nNumberOfSelector, stVariantValues.astLx[nPhase].fTHD_U,         nOFFSET, E_EL3443_Phase.THD_U         );     
    InitSelectorReal(stEL3443MuxReal, nNumberOfSelector, stVariantValues.astLx[nPhase].fRMS_fund_U,    nOFFSET, E_EL3443_Phase.RMS_fund_U    );
    InitSelectorReal(stEL3443MuxReal, nNumberOfSelector, stVariantValues.astLx[nPhase].fF_Ref_U,       nOFFSET, E_EL3443_Phase.F_Ref_U       );
    InitSelectorReal(stEL3443MuxReal, nNumberOfSelector, stVariantValues.astLx[nPhase].fTHD_I,         nOFFSET, E_EL3443_Phase.THD_I        );
    InitSelectorReal(stEL3443MuxReal, nNumberOfSelector, stVariantValues.astLx[nPhase].fTDD_I,         nOFFSET, E_EL3443_Phase.TDD_I        );
    InitSelectorReal(stEL3443MuxReal, nNumberOfSelector, stVariantValues.astLx[nPhase].fRMS_fund_I,    nOFFSET, E_EL3443_Phase.RMS_fund_I   );
    InitSelectorReal(stEL3443MuxReal, nNumberOfSelector, stVariantValues.astLx[nPhase].fF_Ref_I,       nOFFSET, E_EL3443_Phase.F_Ref_I      );
	
    // Initializing the Real Arrays on channel 1 to 3
    FOR i := 0 TO 41 DO
        InitSelectorReal(stEL3443MuxReal, nNumberOfSelector, stVariantValues.astLx[nPhase].fHarmonics_U[i], nOFFSET  + i, E_EL3443_Phase.Harmonics_U);
    END_FOR
    FOR i := 0 TO 41 DO
        InitSelectorReal(stEL3443MuxReal, nNumberOfSelector, stVariantValues.astLx[nPhase].fHarmonics_I[i], nOFFSET  + i, E_EL3443_Phase.Harmonics_I);   
    END_FOR

    // Initializing the ULINT multiplexer on channel 4
    InitSelectorUlint(stEL3443MuxUlint_Ch4, nNumberOfSelectorsCh4, stVariantValues.astLx[nPhase].nU_Last_Zero_Cross, nOFFSET, E_EL3443_Phase.U_Last_Zero_Cross	);
    InitSelectorUlint(stEL3443MuxUlint_Ch4, nNumberOfSelectorsCh4, stVariantValues.astLx[nPhase].nEP,                nOFFSET, E_EL3443_Phase.EP               	);
    InitSelectorUlint(stEL3443MuxUlint_Ch4, nNumberOfSelectorsCh4, stVariantValues.astLx[nPhase].nEP_pos,            nOFFSET, E_EL3443_Phase.EP_pos           	);
    InitSelectorUlint(stEL3443MuxUlint_Ch4, nNumberOfSelectorsCh4, stVariantValues.astLx[nPhase].nEP_neg,            nOFFSET, E_EL3443_Phase.EP_neg           	);
    InitSelectorUlint(stEL3443MuxUlint_Ch4, nNumberOfSelectorsCh4, stVariantValues.astLx[nPhase].nEP_interval,    	 nOFFSET, E_EL3443_Phase.EP_interval     	);
    InitSelectorUlint(stEL3443MuxUlint_Ch4, nNumberOfSelectorsCh4, stVariantValues.astLx[nPhase].nEP_pos_interval,	 nOFFSET, E_EL3443_Phase.EP_pos_interval 	);
    InitSelectorUlint(stEL3443MuxUlint_Ch4, nNumberOfSelectorsCh4, stVariantValues.astLx[nPhase].nEP_neg_interval,	 nOFFSET, E_EL3443_Phase.EP_neg_interval 	);
    InitSelectorUlint(stEL3443MuxUlint_Ch4, nNumberOfSelectorsCh4, stVariantValues.astLx[nPhase].nES,                nOFFSET, E_EL3443_Phase.ES               	);
    InitSelectorUlint(stEL3443MuxUlint_Ch4, nNumberOfSelectorsCh4, stVariantValues.astLx[nPhase].nES_pos,            nOFFSET, E_EL3443_Phase.ES_pos           	);
    InitSelectorUlint(stEL3443MuxUlint_Ch4, nNumberOfSelectorsCh4, stVariantValues.astLx[nPhase].nES_neg,            nOFFSET, E_EL3443_Phase.ES_neg           	);
    InitSelectorUlint(stEL3443MuxUlint_Ch4, nNumberOfSelectorsCh4, stVariantValues.astLx[nPhase].nES_interval,    	 nOFFSET, E_EL3443_Phase.ES_interval     	);
    InitSelectorUlint(stEL3443MuxUlint_Ch4, nNumberOfSelectorsCh4, stVariantValues.astLx[nPhase].nES_pos_interval,	 nOFFSET, E_EL3443_Phase.ES_pos_interval 	);
    InitSelectorUlint(stEL3443MuxUlint_Ch4, nNumberOfSelectorsCh4, stVariantValues.astLx[nPhase].nES_neg_interval,	 nOFFSET, E_EL3443_Phase.ES_neg_interval 	);
    InitSelectorUlint(stEL3443MuxUlint_Ch4, nNumberOfSelectorsCh4, stVariantValues.astLx[nPhase].nEQ,                nOFFSET, E_EL3443_Phase.EQ_              	);
    InitSelectorUlint(stEL3443MuxUlint_Ch4, nNumberOfSelectorsCh4, stVariantValues.astLx[nPhase].nEQ_pos,            nOFFSET, E_EL3443_Phase.EQ_pos           	);
    InitSelectorUlint(stEL3443MuxUlint_Ch4, nNumberOfSelectorsCh4, stVariantValues.astLx[nPhase].nEQ_neg,            nOFFSET, E_EL3443_Phase.EQ_neg           	);
    InitSelectorUlint(stEL3443MuxUlint_Ch4, nNumberOfSelectorsCh4, stVariantValues.astLx[nPhase].nEQ_interval,    	 nOFFSET, E_EL3443_Phase.EQ_interval     	);
    InitSelectorUlint(stEL3443MuxUlint_Ch4, nNumberOfSelectorsCh4, stVariantValues.astLx[nPhase].nEQ_pos_interval,	 nOFFSET, E_EL3443_Phase.EQ_pos_interval 	);
    InitSelectorUlint(stEL3443MuxUlint_Ch4, nNumberOfSelectorsCh4, stVariantValues.astLx[nPhase].nEQ_neg_interval,	 nOFFSET, E_EL3443_Phase.EQ_neg_interval 	);    
END_FOR

// All data that is not assigned to a phase is appended to channels 1 to 4. 

// Real values for multiplexer channel 1   
InitSelectorReal(astEL3443MuxReal_Ch1, nNumberOfSelectorsCh1, stVariantValues.stTotal.fIn_RMS,         E_EL3443_Total.nTotal_OFFSET, E_EL3443_Total.In_RMS        );
InitSelectorReal(astEL3443MuxReal_Ch1, nNumberOfSelectorsCh1, stVariantValues.stTotal.fPower_Factor,   E_EL3443_Total.nTotal_OFFSET, E_EL3443_Total.Power_Factor  );
InitSelectorReal(astEL3443MuxReal_Ch1, nNumberOfSelectorsCh1, stVariantValues.stTotal.fPtot,           E_EL3443_Total.nTotal_OFFSET, E_EL3443_Total.Ptot          );
InitSelectorReal(astEL3443MuxReal_Ch1, nNumberOfSelectorsCh1, stVariantValues.stTotal.fPtotavg,        E_EL3443_Total.nTotal_OFFSET, E_EL3443_Total.Ptotavg       );
InitSelectorReal(astEL3443MuxReal_Ch1, nNumberOfSelectorsCh1, stVariantValues.stTotal.fPtotmin,        E_EL3443_Total.nTotal_OFFSET, E_EL3443_Total.Ptotmin       );
InitSelectorReal(astEL3443MuxReal_Ch1, nNumberOfSelectorsCh1, stVariantValues.stTotal.fPtotmax,        E_EL3443_Total.nTotal_OFFSET, E_EL3443_Total.Ptotmax       );
InitSelectorReal(astEL3443MuxReal_Ch1, nNumberOfSelectorsCh1, stVariantValues.stTotal.fStot,           E_EL3443_Total.nTotal_OFFSET, E_EL3443_Total.Stot          );

// Real values for multiplexer channel 2
InitSelectorReal(astEL3443MuxReal_Ch2, nNumberOfSelectorsCh2, stVariantValues.stTotal.fStotavg,   E_EL3443_Total.nTotal_OFFSET, E_EL3443_Total.Stotavg);                                                                                                                        
InitSelectorReal(astEL3443MuxReal_Ch2, nNumberOfSelectorsCh2, stVariantValues.stTotal.fStotmin,   E_EL3443_Total.nTotal_OFFSET, E_EL3443_Total.Stotmin);
InitSelectorReal(astEL3443MuxReal_Ch2, nNumberOfSelectorsCh2, stVariantValues.stTotal.fStotmax,   E_EL3443_Total.nTotal_OFFSET, E_EL3443_Total.Stotmax);
InitSelectorReal(astEL3443MuxReal_Ch2, nNumberOfSelectorsCh2, stVariantValues.stTotal.fQtot,      E_EL3443_Total.nTotal_OFFSET, E_EL3443_Total.Qtot   );
InitSelectorReal(astEL3443MuxReal_Ch2, nNumberOfSelectorsCh2, stVariantValues.stTotal.fQtotavg,   E_EL3443_Total.nTotal_OFFSET, E_EL3443_Total.Qtotavg);
InitSelectorReal(astEL3443MuxReal_Ch2, nNumberOfSelectorsCh2, stVariantValues.stTotal.fQtotmin,   E_EL3443_Total.nTotal_OFFSET, E_EL3443_Total.Qtotmin);
InitSelectorReal(astEL3443MuxReal_Ch2, nNumberOfSelectorsCh2, stVariantValues.stTotal.fQtotmax,   E_EL3443_Total.nTotal_OFFSET, E_EL3443_Total.Qtotmax);

//Real values for multiplexer channel 3
InitSelectorReal(astEL3443MuxReal_Ch3, nNumberOfSelectorsCh3, stVariantValues.stTotal.fPhiL1L2,   E_EL3443_Total.nTotal_OFFSET, E_EL3443_Total.PhiL1L2  );
InitSelectorReal(astEL3443MuxReal_Ch3, nNumberOfSelectorsCh3, stVariantValues.stTotal.fPhiL1L3,   E_EL3443_Total.nTotal_OFFSET, E_EL3443_Total.PhiL1L3  );
InitSelectorReal(astEL3443MuxReal_Ch3, nNumberOfSelectorsCh3, stVariantValues.stTotal.fUnbalance, E_EL3443_Total.nTotal_OFFSET, E_EL3443_Total.Unbalance);
InitSelectorReal(astEL3443MuxReal_Ch3, nNumberOfSelectorsCh3, stVariantValues.stTotal.fPQF,       E_EL3443_Total.nTotal_OFFSET, E_EL3443_Total.PQF      );
InitSelectorReal(astEL3443MuxReal_Ch3, nNumberOfSelectorsCh3, stVariantValues.stTotal.fPQF_Avg,   E_EL3443_Total.nTotal_OFFSET, E_EL3443_Total.PQF_Avg  );
InitSelectorReal(astEL3443MuxReal_Ch3, nNumberOfSelectorsCh3, stVariantValues.stTotal.fPQF_Min,   E_EL3443_Total.nTotal_OFFSET, E_EL3443_Total.PQF_MIN  );
InitSelectorReal(astEL3443MuxReal_Ch3, nNumberOfSelectorsCh3, stVariantValues.stTotal.fPQF_Max,   E_EL3443_Total.nTotal_OFFSET, E_EL3443_Total.PQF_MAX);


// Ulint values for multiplexer channel 4
InitSelectorUlint(stEL3443MuxUlint_Ch4, nNumberOfSelectorsCh4, stVariantValues.stTotal.nEptot,                    E_EL3443_Total.nTotal_OFFSET, E_EL3443_Total.Eptot           	);
InitSelectorUlint(stEL3443MuxUlint_Ch4, nNumberOfSelectorsCh4, stVariantValues.stTotal.nEPtot_pos,                E_EL3443_Total.nTotal_OFFSET, E_EL3443_Total.EPtot_pos        );
InitSelectorUlint(stEL3443MuxUlint_Ch4, nNumberOfSelectorsCh4, stVariantValues.stTotal.nEPtot_neg,                E_EL3443_Total.nTotal_OFFSET, E_EL3443_Total.EPtot_neg        );
InitSelectorUlint(stEL3443MuxUlint_Ch4, nNumberOfSelectorsCh4, stVariantValues.stTotal.nEptot_interval,          E_EL3443_Total.nTotal_OFFSET, E_EL3443_Total.Eptot_interval    );
InitSelectorUlint(stEL3443MuxUlint_Ch4, nNumberOfSelectorsCh4, stVariantValues.stTotal.nEPtot_pos_interval,      E_EL3443_Total.nTotal_OFFSET, E_EL3443_Total.EPtot_pos_interval);
InitSelectorUlint(stEL3443MuxUlint_Ch4, nNumberOfSelectorsCh4, stVariantValues.stTotal.nEPtot_neg_interval,      E_EL3443_Total.nTotal_OFFSET, E_EL3443_Total.EPtot_neg_interval);
InitSelectorUlint(stEL3443MuxUlint_Ch4, nNumberOfSelectorsCh4, stVariantValues.stTotal.nEStot,                    E_EL3443_Total.nTotal_OFFSET, E_EL3443_Total.EStot            );
InitSelectorUlint(stEL3443MuxUlint_Ch4, nNumberOfSelectorsCh4, stVariantValues.stTotal.nEStot_pos,                E_EL3443_Total.nTotal_OFFSET, E_EL3443_Total.EStot_pos        );
InitSelectorUlint(stEL3443MuxUlint_Ch4, nNumberOfSelectorsCh4, stVariantValues.stTotal.nEStot_neg,                E_EL3443_Total.nTotal_OFFSET, E_EL3443_Total.EStot_neg        );
InitSelectorUlint(stEL3443MuxUlint_Ch4, nNumberOfSelectorsCh4, stVariantValues.stTotal.nEStot_interval,          E_EL3443_Total.nTotal_OFFSET, E_EL3443_Total.EStot_interval    );
InitSelectorUlint(stEL3443MuxUlint_Ch4, nNumberOfSelectorsCh4, stVariantValues.stTotal.nEStot_pos_interval,      E_EL3443_Total.nTotal_OFFSET, E_EL3443_Total.EStot_pos_interval);
InitSelectorUlint(stEL3443MuxUlint_Ch4, nNumberOfSelectorsCh4, stVariantValues.stTotal.nEStot_neg_interval,      E_EL3443_Total.nTotal_OFFSET, E_EL3443_Total.EStot_neg_interval);
InitSelectorUlint(stEL3443MuxUlint_Ch4, nNumberOfSelectorsCh4, stVariantValues.stTotal.nEQtot,                    E_EL3443_Total.nTotal_OFFSET, E_EL3443_Total.EQtot            );
InitSelectorUlint(stEL3443MuxUlint_Ch4, nNumberOfSelectorsCh4, stVariantValues.stTotal.nEQtot_pos,                E_EL3443_Total.nTotal_OFFSET, E_EL3443_Total.EQtot_pos        );
InitSelectorUlint(stEL3443MuxUlint_Ch4, nNumberOfSelectorsCh4, stVariantValues.stTotal.nEQtot_neg,                E_EL3443_Total.nTotal_OFFSET, E_EL3443_Total.EQtot_neg        );
InitSelectorUlint(stEL3443MuxUlint_Ch4, nNumberOfSelectorsCh4, stVariantValues.stTotal.nEQtot_interval,          E_EL3443_Total.nTotal_OFFSET, E_EL3443_Total.EQtot_interval    );
InitSelectorUlint(stEL3443MuxUlint_Ch4, nNumberOfSelectorsCh4, stVariantValues.stTotal.nEQtot_pos_interval,      E_EL3443_Total.nTotal_OFFSET, E_EL3443_Total.EQtot_pos_interval);
InitSelectorUlint(stEL3443MuxUlint_Ch4, nNumberOfSelectorsCh4, stVariantValues.stTotal.nEQtot_neg_interval,      E_EL3443_Total.nTotal_OFFSET, E_EL3443_Total.EQtot_neg_interval);
END_METHOD

(*This method calculates the selector based on the offset and the base selector and sets the corresponding reference*)
METHOD PRIVATE InitSelectorReal : HRESULT
VAR_IN_OUT
    stEL3443MuxReal : ARRAY [0..nARRAYSIZEMUXREAL] OF ST_EL3443_MUX_REAL;
    nNumberOfSelectors : UINT;    
    fValue : REAL;  
END_VAR
VAR_INPUT
    nOFFSET : UINT;
    nSelector : UINT;
END_VAR
    stEL3443MuxReal[nNumberOfSelectors].nSelector := nSelector + nOFFSET; //Basis Selector + Channel(Phase) Offset
    stEL3443MuxReal[nNumberOfSelectors].fValueRef REF= fValue; //Set reference to create a link between selector and output value
    nNumberOfSelectors := nNumberOfSelectors + 1;
END_METHOD

(*This method calculates the selector based on the offset and the base selector and sets the corresponding pointer address*)
METHOD PRIVATE InitSelectorUlint : HRESULT
VAR_IN_OUT
    stEL3443MuxUlint : ARRAY [0..nARRAYSIZEMUXULINT] OF ST_EL3443_MUX_ULINT;
    nNumberOfSelectors : UINT;      
END_VAR
VAR_INPUT
    nValue : ANY_INT;
    nOFFSET : UINT;
    nSelector : UINT;
END_VAR
    stEL3443MuxUlint[nNumberOfSelectors].nSelector := nSelector + nOFFSET; //Basis Selector + Channel(Phase) Offset
    stEL3443MuxUlint[nNumberOfSelectors].nValueRef := nValue.pValue; //Set reference to create a link between selector and output value
    nNumberOfSelectors := nNumberOfSelectors + 1;
END_METHOD

END_FUNCTION_BLOCK
